Yaskawa INFORM job: DEMO.JBI

/JOB
//NAME DEMO
//POS
///NPOS 3,0,0,0
///TOOL 0
///PULSE
C000=-4720,45472,-31419,-53,8048,2945
C001=-4720,49552,-31419,-53,8048,2945
C002=-1264,43504,-30699,-53,8048,2945
//INST
///DATE 2014/11/04 13:48
///ATTR 0,0,0,0,0,0,0,0,0,0,0,0,0,1,0,0
///FRAME BASE
NOP
*1
MOVL C000 V=11.7 CONT
MOVJ C001 VJ=1.00 CONT
MOVJ C002 VJ=0.78 CONT
JUMP *1
END
